Staubli VAL3: getStatus.pgx

public program getStatus(num x_nConvNum, num& x_nStatus[])
  local bool l_bQuit
  local bool l_bLock
  local num l_i
  local num l_nStatus
  local num l_nStep
  local string l_sSubString
begin
  // This program returns the status of the conveyor library
  //
  // Input Param
  // x_nConvNum    : Conveyor Number
  //
  // Output Param
  //  x_nStatus    : Status of the conveyor library
  //
  //Created 04-06-07                              C.CURRIVAND
  //--------------------------------------------------------------
  //
  l_bQuit=false
  do
    switch l_nStep
      // Check status of the encoder library
      case 0
        call enc:getStatus(l_nStatus)
        if (l_nStatus!=0)
          // Prepare clear text error message
          call ut:addNumToString(sErrMsgList[7],sErrorMessage,"",l_nStatus)
          l_bQuit=true
        else
          l_nStep=20
        endIf
      break
      // Check status of the detection library.
      case 10
        //call det:getStatus(l_nStatus)
        if (l_nStatus!=0)
          // Prepare clear text error message
          call ut:addNumToString(sErrMsgList[8],sErrorMessage,"",l_nStatus)
          l_bQuit=true
        else
          l_nStep=20
        endIf
      break
      // check status of the conveyor task
      // sTASK[0]=conveyor
      case 20
        l_nStatus=taskStatus(sTASK[0]+toString("",x_nConvNum))
        if (l_nStatus!=0) and (l_nStatus!=1)
          // Prepare clear text error message
          if l_nStatus==-1
            // Task not created (yet !)
            l_nStatus=2999
          else
            // Run-time error
            l_nStatus=2000+l_nStatus
          endIf
          l_sSubString=sTASK[0]+toString("",x_nConvNum)
          call ut:addStrToString(sErrMsgList[6],sErrorMessage,"",l_sSubString)
          call ut:addNumToString(sErrorMessage,sErrorMessage,"*",l_nStatus)
          l_bQuit=true
        endIf
        if (l_nStatus==0) or (l_nStatus==1)
          l_nStatus=nStatus
          nStatus=0
        endIf
        l_bQuit=true
      break
    endSwitch
    delay(0)
  until l_bQuit==true
  x_nStatus=l_nStatus
end
